(* IEC 61131-3 sources: AxisLib/src/MappAr/MotionControl/AxisBasic, 6 files *)

(* ---- AxisBasic.typ ---- *)
(*
* File: Types.typ
* Copyright (c) 2023 Loupe
* https://loupe.team
*
* This file is part of AxisLib, licensed under the MIT License.
*
*)

TYPE
	Configuration_typ : 	STRUCT
		Axis : ARRAY[0..MAI_AXIS]OF AxisConfiguration_typ;
		velocity : REAL;
		acceleration : REAL;
		deceleration : REAL;
	END_STRUCT;
	AxisConfiguration_typ : 	STRUCT
		power : BOOL;
		cfg : AxisBasic_IN_CFG_typ;
	END_STRUCT;
	Task_typ : 	STRUCT
		cmd : Task_Cmd_typ;
		parameters : AxisBasic_IN_PAR_typ;
		status : Task_Status_typ;
		internal : Task_Internal_typ;
	END_STRUCT;
	Task_Cmd_typ : 	STRUCT
		New_Member : BOOL;
	END_STRUCT;
	Task_Status_typ : 	STRUCT
		state : ARRAY[0..MAI_AXIS]OF State_enum;
		axisError : ARRAY[0..MAI_AXIS]OF BOOL;
		axisErrorReset : ARRAY[0..MAI_AXIS]OF BOOL;
	END_STRUCT;
	Task_Internal_typ : 	STRUCT
		axisInternal : ARRAY[0..MAI_AXIS]OF AxisBasic_Internal_typ;
		MC_MoveVelocity : ARRAY[0..MAI_AXIS]OF MC_MoveVelocity;
	END_STRUCT;
	(*Sim_typ : 	STRUCT
		axisMoving : ARRAY[0..MAI_AXIS]OF BOOL;
	END_STRUCT;*)
	State_enum :
		(
		ST_POWER_ON,
		ST_MOVE_VELOCITY,
		ST_ERROR
		);

END_TYPE

(* ---- AxisBasic.st ---- *)
(*
* File: Types.typ
* Copyright (c) 2023 Loupe
* https://loupe.team
*
* This file is part of AxisLib, licensed under the MIT License.
*
*)

(********************************************************************
This task defines the behavior of the axes in the system. Axes begin
motion in the excute piper state. Stop triggers a graceful stop (i.e.
finish what your doing and then stop) with the inverters still
powered on (recoverable). Abort triggers an immediate stop of the
axes with the inverters powered off (unrecoverable). Axis errors are
collected in execute and idle and can be reset without effecting
other axes.
********************************************************************)
PROGRAM _INIT

	AxisConfig;

END_PROGRAM

PROGRAM _CYCLIC

	// Piper
	PiperModuleInterface;

	FOR axisIdx := 0 TO MAI_AXIS DO

		gMotorBasic[axisIdx].IN.PAR.Acceleration := Configuration.acceleration;
		gMotorBasic[axisIdx].IN.PAR.Deceleration := Configuration.deceleration;
		gMotorBasic[axisIdx].IN.PAR.Velocity := Configuration.velocity;

		// cyclically call axis basic
		AxisBasicCyclic(gMotorBasic[axisIdx], Configuration.Axis[axisIdx].cfg, task.internal.axisInternal[axisIdx]);

		//sim.axisMoving[axisIdx] := gMotorBasic[axisIdx].OUT.PLCOpenDiscrete.ContinuousMotion;

	END_FOR

	// reset commands
	FOR axisIdx := 0 TO MAI_AXIS DO
		task.status.axisErrorReset[axisIdx] := FALSE;
		gMotorBasic[axisIdx].IN.CMD.MoveVelocity := FALSE;
		gMotorBasic[axisIdx].IN.CMD.ErrorReset := FALSE;
	END_FOR

END_PROGRAM

(* ---- AxisConfig.st ---- *)
(*
* File: Types.typ
* Copyright (c) 2023 Loupe
* https://loupe.team
*
* This file is part of AxisLib, licensed under the MIT License.
*
*)

ACTION AxisConfig:

	// Assign axis pointers.
	gMotorBasic[Axis_1].pAxisObject := ADR(gAxis_1);
	gMotorBasic[Axis_2].pAxisObject := ADR(gAxis_2);
	gMotorBasic[Axis_3].pAxisObject := ADR(gAxis_3);
	gMotorBasic[Axis_4].pAxisObject := ADR(gAxis_4);

END_ACTION

(* ---- PiperInterface.st ---- *)
(*
* File: Types.typ
* Copyright (c) 2023 Loupe
* https://loupe.team
*
* This file is part of AxisLib, licensed under the MIT License.
*
*)

(*
The intent for this piper implementation is to power on and move velocity
all the axes in execute, respond to errors in execute without the need for
system wide abort/reset, and allow enabling/disabling of axes at runtime.
*)
ACTION PiperModuleInterface:

	//Give this module a name so it is easier to debug
	ModuleInterface.ModuleName:=	'AxisMgr';
	// cyclically clear ModuleStatus so we don't have to worry about clearing it when states change
	brsmemset(ADR(ModuleInterface.ModuleStatus), 0, SIZEOF(ModuleInterface.ModuleStatus));

	//Add a module to the Piper
	Module.ModuleInterface:=	ADR(ModuleInterface);
	Module.Piper:= 	ADR(gMachine);
	Module();

	// Handle any machine states that this module needs to respond to
	CASE ModuleInterface.PiperState OF
		MACH_ST_BOOTING: // Wait for axes to come on line (CommunicationReady) and restore position

			CASE ModuleInterface.PiperSubState OF

				SUB_STATE_INIT:
					ModuleInterface.ModuleSubStateRequest := SUB_STATE_BOOTING_COMM_READY;

				SUB_STATE_BOOTING_COMM_READY:
					groupStatus := TRUE;
					ModuleInterface.ModuleStatus := 'Waiting on axis:';

					FOR axisIdx := 0 TO MAI_AXIS DO
						IF Configuration.Axis[axisIdx].cfg.Active THEN
							IF gMotorBasic[axisIdx].OUT.PLCOpenDiscrete.Errorstop THEN
								// let axis pass through
							ELSIF NOT gMotorBasic[axisIdx].OUT.State.CommunicationReady THEN
								groupStatus := FALSE;
								ModuleInterface.ModuleStatus := CONCAT(ModuleInterface.ModuleStatus, CONCAT(gMotorBasic[axisIdx].OUT.Name,' '));
							END_IF
						END_IF
					END_FOR

					IF groupStatus THEN
						ModuleInterface.ModuleResponse := ModuleInterface.PiperState;
					END_IF

			END_CASE

		MACH_ST_CLEARING:
			groupStatus := TRUE;
			FOR axisIdx := 0 TO MAI_AXIS DO
				IF gMotorBasic[axisIdx].OUT.ErrorCount > 0 THEN
					groupStatus := FALSE;
					gMotorBasic[axisIdx].IN.CMD.ErrorReset := TRUE;
				END_IF
			END_FOR

			IF groupStatus THEN
				ModuleInterface.ModuleResponse := ModuleInterface.PiperState;
			END_IF

		//MACH_ST_STOPPED:
		//MACH_ST_STARTING:
		MACH_ST_IDLE,
		//MACH_ST_SUSPENDED:
//		MACH_ST_EXECUTE:
//
//			FOR axisIdx := 0 TO MAI_AXIS DO
//
//				IF gMotorBasic[axisIdx].OUT.ErrorCount > 0 THEN
//					task.status.state[axisIdx] := ST_ERROR;
//				END_IF
//
//				CASE task.status.state[axisIdx] OF
//
//					ST_POWER_ON:
//
//						gMotorBasic[axisIdx].IN.CMD.Power := TRUE;
//						IF gMotorBasic[axisIdx].OUT.State.PowerOn AND (gMachine.OUT.State = MACH_ST_EXECUTE) THEN
//							task.status.state[axisIdx] := ST_MOVE_VELOCITY;
//						END_IF
//
//					ST_MOVE_VELOCITY:
//
//						IF Configuration.Axis[axisIdx].cfg.Active AND Configuration.Axis[axisIdx].power THEN
//							gMotorBasic[axisIdx].IN.CMD.MoveVelocity := TRUE;
//						END_IF
//
//					ST_ERROR:
//
//						task.status.axisError[axisIdx] := TRUE;
//						gMotorBasic[axisIdx].IN.CMD.ErrorReset := task.status.axisErrorReset[axisIdx];
//						IF gMotorBasic[axisIdx].OUT.ErrorCount = 0 THEN
//							task.status.state[axisIdx] := ST_POWER_ON;
//						END_IF
//
//				END_CASE
//
//			END_FOR

		MACH_ST_STOPPING:

			CASE ModuleInterface.PiperSubState OF

				SUB_STATE_INIT:
					ModuleInterface.ModuleSubStateRequest := SUB_STATE_STOP;

				SUB_STATE_STOP:
					groupStatus := TRUE;
					ModuleInterface.ModuleStatus := 'Stopping axis:';

					FOR axisIdx := 0 TO MAI_AXIS DO
						IF Configuration.Axis[axisIdx].cfg.Active AND Configuration.Axis[axisIdx].power THEN
							gMotorBasic[axisIdx].IN.CMD.Stop := gMotorBasic[axisIdx].OUT.PLCOpenDiscrete.ContinuousMotion
																OR gMotorBasic[axisIdx].OUT.PLCOpenDiscrete.DiscreteMotion
																OR gMotorBasic[axisIdx].OUT.PLCOpenDiscrete.Homing
																OR gMotorBasic[axisIdx].OUT.PLCOpenDiscrete.SynchronizedMotion;
							IF gMotorBasic[axisIdx].OUT.PLCOpenDiscrete.Errorstop THEN
								// let axis pass through
							ELSIF gMotorBasic[axisIdx].IN.CMD.Stop OR gMotorBasic[axisIdx].OUT.PLCOpenDiscrete.Stopping THEN
								groupStatus := FALSE;
								ModuleInterface.ModuleStatus := CONCAT(ModuleInterface.ModuleStatus, CONCAT(gMotorBasic[axisIdx].OUT.Name,' '));
							END_IF
						END_IF
					END_FOR

					IF groupStatus THEN
						ModuleInterface.ModuleResponse := ModuleInterface.PiperState;
					END_IF

			END_CASE

		MACH_ST_ABORTING:

			CASE ModuleInterface.PiperSubState OF

				SUB_STATE_INIT:
					ModuleInterface.ModuleSubStateRequest := SUB_STATE_STOP;

				SUB_STATE_STOP:
					groupStatus := TRUE;
					ModuleInterface.ModuleStatus := 'Stopping axis:';

					FOR axisIdx := 0 TO MAI_AXIS DO
						IF Configuration.Axis[axisIdx].cfg.Active AND Configuration.Axis[axisIdx].power THEN
							gMotorBasic[axisIdx].IN.CMD.Stop := gMotorBasic[axisIdx].OUT.PLCOpenDiscrete.ContinuousMotion
																OR gMotorBasic[axisIdx].OUT.PLCOpenDiscrete.DiscreteMotion
																OR gMotorBasic[axisIdx].OUT.PLCOpenDiscrete.Homing
																OR gMotorBasic[axisIdx].OUT.PLCOpenDiscrete.SynchronizedMotion;
							IF gMotorBasic[axisIdx].OUT.PLCOpenDiscrete.Errorstop THEN
								// let axis pass through
							ELSIF gMotorBasic[axisIdx].IN.CMD.Stop OR gMotorBasic[axisIdx].OUT.PLCOpenDiscrete.Stopping THEN
								groupStatus := FALSE;
								ModuleInterface.ModuleStatus := CONCAT(ModuleInterface.ModuleStatus, CONCAT(gMotorBasic[axisIdx].OUT.Name,' '));
							END_IF
						END_IF
					END_FOR

					IF groupStatus THEN
						ModuleInterface.ModuleSubStateRequest := SUB_STATE_ABORTING_POWER_OFF;
					END_IF

				SUB_STATE_ABORTING_POWER_OFF:
					groupStatus := TRUE;
					ModuleInterface.ModuleStatus := 'Powering Off axis:';

					FOR axisIdx := 0 TO MAI_AXIS DO
						IF Configuration.Axis[axisIdx].power THEN
							gMotorBasic[axisIdx].IN.CMD.Power := FALSE;
							IF gMotorBasic[axisIdx].OUT.PLCOpenDiscrete.Errorstop THEN
								// let axis pass through
							ELSIF NOT gMotorBasic[axisIdx].OUT.PLCOpenDiscrete.Disabled THEN
								groupStatus := FALSE;
								ModuleInterface.ModuleStatus := CONCAT(ModuleInterface.ModuleStatus, CONCAT(gMotorBasic[axisIdx].OUT.Name,' '));
							END_IF
						END_IF
					END_FOR

					IF groupStatus THEN
						ModuleInterface.ModuleResponse := ModuleInterface.PiperState;
					END_IF

			END_CASE

		//MACH_ST_ABORTED:
		//MACH_ST_HOLDING:
		//MACH_ST_HELD:
		//MACH_ST_UNHOLDING:
		//MACH_ST_SUSPENDING:
		//MACH_ST_UNSUSPENDING:
		MACH_ST_RESETTING:

			CASE ModuleInterface.PiperSubState OF

				SUB_STATE_INIT:
					ModuleInterface.ModuleSubStateRequest := SUB_STATE_RESETTING_POWER_ON;

				SUB_STATE_RESETTING_POWER_ON:
					groupStatus := TRUE;
					ModuleInterface.ModuleStatus := 'Powering on axis:';

					FOR axisIdx := 0 TO MAI_AXIS DO
						task.status.state[axisIdx] := ST_POWER_ON;
						IF Configuration.Axis[axisIdx].cfg.Active AND Configuration.Axis[axisIdx].power THEN
							IF gMotorBasic[axisIdx].OUT.PLCOpenDiscrete.Errorstop THEN
								// let axis pass through
							ELSIF NOT gMotorBasic[axisIdx].OUT.State.PowerOn THEN
								groupStatus := FALSE;
								gMotorBasic[axisIdx].IN.CMD.Power := TRUE;
								ModuleInterface.ModuleStatus := CONCAT(ModuleInterface.ModuleStatus, CONCAT(gMotorBasic[axisIdx].OUT.Name,' '));
							END_IF
						END_IF
					END_FOR

					IF groupStatus THEN
						ModuleInterface.ModuleResponse := ModuleInterface.PiperState;
					END_IF

			END_CASE

		//MACH_ST_COMPLETING:
		//MACH_ST_COMPLETE:
		//MACH_ST_BYPASSED:

		ELSE
			ModuleInterface.ModuleResponse:=	ModuleInterface.PiperState;

	END_CASE

END_ACTION

(* ---- PiperModule.var ---- *)
(*
* File: Types.typ
* Copyright (c) 2023 Loupe
* https://loupe.team
*
* This file is part of AxisLib, licensed under the MIT License.
*
*)

VAR
	ModuleInterface : Module_Interface_typ;
	Module : Piper_Module_Fub;
END_VAR

(* ---- AxisBasic.var ---- *)
(*
* File: Types.typ
* Copyright (c) 2023 Loupe
* https://loupe.team
*
* This file is part of AxisLib, licensed under the MIT License.
*
*)

VAR
	Configuration : Configuration_typ;
	groupStatus : BOOL;
	axisIdx : UDINT;
	task : Task_typ;
(*	sim : Sim_typ;*)
END_VAR
